PROGRAM MAIN
VAR
	fbExtTimeSoft : FB_TcExternalTime(ExternalTimeSoft);
	fbSender: FB_MUDPI_SENDER;
	payload: T_PAYLOAD;
	fbTimer: FB_TIME;
	
END_VAR

fbTimer();
fbSender();
payload.data1 := payload.data1 + 1;
fbSender.SetTimestamp(fbTimer.GetMudpiTime());
fbSender.SetMudpiPayload(ADR(payload), SIZEOF(payload));
fbSender.SendData();

END_PROGRAM

(* stored: Version 1.1.0.1, ProductVersion 3.1.4024.9
   POU MAIN: Id {a54cb7a1-7b45-44b3-b235-145807ae3efc}, SpecialFunc None *)
